{attribute 'linkalways'} 
{attribute 'no_explicit_call' := 'This FB is a CLASS and must be accessed using methods or properties'}
{attribute 'enable_dynamic_creation'}
FUNCTION_BLOCK _LINT EXTENDS NumericDatatypeBase
VAR
	localData : LINT;
	activeData : REFERENCE TO LINT REF= localData;
END_VAR

PROPERTY PUBLIC Address : PVOID
GET
Address := ADR(activeData);
END_GET
END_PROPERTY

METHOD PUBLIC ClearReference
VAR_INPUT
END_VAR
activeData REF= localData;
END_METHOD

METHOD PUBLIC Clone : I_Datatype
VAR
    pClone : POINTER TO _LINT;
END_VAR
pClone := __NEW(_LINT(InitialValue := Value));
Clone := pClone^;
END_METHOD

METHOD FB_init : BOOL
VAR_INPUT
	bInitRetains : BOOL; // if TRUE, the retain variables are initialized (warm start / cold start)
	bInCopyCode : BOOL;  // if TRUE, the instance afterwards gets moved into the copy code (online change)
	InitialValue : LINT;
END_VAR
localData := InitialValue;
END_METHOD

PROPERTY PUBLIC IsFloat : BOOL
GET
IsFloat := FALSE;
END_GET
END_PROPERTY

PROPERTY PUBLIC IsSigned : BOOL
GET
IsSigned := TRUE;
END_GET
END_PROPERTY

METHOD PUBLIC MakeReferenceTo
VAR_INPUT
	ReferenceTarget : REFERENCE TO LINT;
END_VAR
activeData REF= ReferenceTarget;
END_METHOD

PROPERTY PUBLIC MaxValue : LINT
GET
MaxValue :=  DatatypeLimits.LINT_MAX_VALUE;
END_GET
END_PROPERTY

PROPERTY PUBLIC MinValue : LINT
GET
MinValue := DatatypeLimits.LINT_MIN_VALUE;
END_GET
END_PROPERTY

METHOD PROTECTED SerializeMaxValue
VAR_INPUT
	Serializer : I_Serializer;
END_VAR
Serializer.AddLint(MaxValue);
END_METHOD

METHOD PROTECTED SerializeMinValue
VAR_INPUT
	Serializer : I_Serializer;
END_VAR
Serializer.AddLint(MinValue);
END_METHOD

METHOD PUBLIC SerializeWith
VAR_INPUT
	Serializer : I_Serializer;
END_VAR
Serializer.AddLint(activeData);
END_METHOD

PROPERTY PUBLIC Size : UDINT
GET
Size := SIZEOF(activeData);
END_GET
END_PROPERTY

METHOD TryDeserializeFrom : BOOL
VAR_INPUT
	Deserializer : I_Deserializer;
	Feedback : I_DeserializerFeedback;
END_VAR
TryDeserializeFrom := Deserializer.TryGetLint(activeData, Feedback);
END_METHOD

METHOD TryMakeReferenceTo : BOOL
VAR_INPUT
	Target : I_Datatype;
END_VAR
VAR
	pTargetData : POINTER TO LINT;
END_VAR
IF NOT (Target.TypeName = TypeName) THEN
	RETURN;
END_IF

pTargetData := Target.Address;
activeData REF= pTargetData^;
TryMakeReferenceTo := TRUE;
END_METHOD

PROPERTY PUBLIC TypeName : T_MAXSTRING
GET
TypeName := 'LINT';
END_GET
END_PROPERTY

PROPERTY PUBLIC Value : LINT
GET
Value := activeData;
END_GET
SET
activeData := Value;
END_SET
END_PROPERTY

END_FUNCTION_BLOCK

(* stored: Version 1.1.0.1, ProductVersion 3.1.4024.12
   POU _LINT: Id {17b89840-9ab0-0782-1caf-fbb224dd5313}, SpecialFunc None
   Folder Constructor: Id {e75c475d-cb92-0fbe-180d-78c14019c391}
   Folder Protected: Id {3b3d2a91-a940-00be-3f54-1712e5f6b68a}
   Property Address: Id {4c80cab2-f3a8-0698-268c-94c78bc601e2}
   Get Get: Id {7ff5e8fc-9243-0fa3-01e4-cc0ba8106d8f}
   Method ClearReference: Id {47c3693b-2562-0e0a-1565-af858bfb28f1}
   Method Clone: Id {ec9e86ba-e052-058f-1273-2dec5a50675b}
   Method FB_init: Id {6f5bef10-04cb-0b63-34bb-4c3669166cf6}
   Property IsFloat: Id {ad49b7b4-4ed2-04be-3965-eefae1919961}
   Get Get: Id {a5bab67e-9d51-03ed-19ac-bc64b4f9973b}
   Property IsSigned: Id {a931b414-132e-06f4-267c-3b9fab46d244}
   Get Get: Id {46e6e594-2a63-01f7-10f0-12f09e63402a}
   Method MakeReferenceTo: Id {2c209dec-5b56-0d45-2e4e-964832defbed}
   Property MaxValue: Id {048a600b-5ea0-0e97-2cfe-a4c5fc2ba388}
   Get Get: Id {f51c3fbe-9b78-0bbd-080e-9ac73e20a908}
   Property MinValue: Id {184f8e42-c0dd-0a28-25f7-c17b21372b1c}
   Get Get: Id {ed90aa3c-614c-0ff3-3062-9679398b6d21}
   Method SerializeMaxValue: Id {b8680d96-233c-0731-012d-c274bb4ff48e}
   Method SerializeMinValue: Id {30eca15f-9ba5-08de-0b7a-d3ccc06ffbb9}
   Method SerializeWith: Id {4cf4b3ba-a687-0979-165c-ca7c26df1014}
   Property Size: Id {798063c9-e1ab-0f08-2d92-fdb7efa97a69}
   Get Get: Id {ce3da064-d59e-0d53-220e-8e933d765f82}
   Method TryDeserializeFrom: Id {aa3a6ab6-ca0c-0b44-3f04-30766dec01c1}
   Method TryMakeReferenceTo: Id {42e5f4a3-a405-092d-3cee-0cfc6d827e13}
   Property TypeName: Id {adfa31e0-80dd-022e-211b-64ddad620d23}
   Get Get: Id {79917b27-c73a-01a9-3b99-3b3ebdc61393}
   Property Value: Id {c5f146c2-3d68-0487-2e7d-78e3f0c64513}
   Get Get: Id {7295dd5e-7b28-0811-11cc-f10e0c042d4a}
   Set Set: Id {8a41e9bb-1c33-0e8b-1a87-71f8b042af57} *)
